// TIA Portal V17 export
// export: Created 2025-03-13T10:31:00.8297075Z, ExportSetting WithDefaults, DisplayName Totally Integrated Automation Portal, DisplayVersion V17 Update 8, DisplayName TIA Portal Openness, DisplayVersion V17 Update 8, DisplayName TIA Portal Version Control Interface, DisplayVersion V17, DisplayName SINAMICS Startdrive Advanced, DisplayVersion V17 SP2, DisplayName SINAMICS Startdrive G110M, G120, G120C, G120D, G120P, G115D, DisplayVersion V17 SP2, DisplayName SINAMICS Startdrive G130, G150, S120, S150, SINAMICS MV, S210, DisplayVersion V17 SP2, DisplayName STEP 7 Professional, DisplayVersion V17 Update 8, DisplayName SINUMERIK ONE STEP 7 Toolbox, DisplayVersion V17 Update 12, DisplayName SINUMERIK 840D sl STEP 7 Toolbox, DisplayVersion V17 Update 12, DisplayName STEP 7 Safety, DisplayVersion V17 Update 6, DisplayName WinCC Advanced, DisplayVersion V17 Update 8
DATA_BLOCK "LTLP_SLDiagnosticToIdentDB"   // DB592
{ DB_Accessible_From_OPC_UA := 'FALSE' }
// stored: AutoNumber true, DBAccessibleFromOPCUA false, DBAccessibleFromWebserver true, InstanceOfName LTLP_SLDiagnosticToIdent, InstanceOfType FB
"LTLP_SLDiagnosticToIdent"
   // VAR_INPUT
   //    ENABLE : Bool;
   //    ResetReaderDone : Bool;
   //    ReadReaderDone : Bool;
   //    SetReaderDone : Bool;
   //    StateOfDoneCmd : DWord;
   //    DeviceIdent : TO_IDENT;
   // END_VAR
   // VAR
   //    stDiagnosticData { S7_SetPoint := 'True'} : "LTLP_typeDiagnosticIdent";
   // END_VAR
BEGIN
END_DATA_BLOCK
